FUNCTION_BLOCK CheckStatus
VAR_INPUT
	Position :INT;
	InputArray: ARRAY [1..25] OF BOOL;
END_VAR
VAR_OUTPUT
Occupied : BOOL;
END_VAR

Occupied := FALSE;
IF InputArray[Position] THEN
	Occupied := TRUE;
END_IF

END_FUNCTION_BLOCK

(* stored: Version 1.1.0.1, ProductVersion 3.1.4022.12
   POU CheckStatus: Id {c3ef0c3f-40cd-4ce4-a305-43916db7ede3}, SpecialFunc None *)
